// TIA Portal V20 export
// export: Created 2026-09-14T11:29:01.3083632Z, ExportSetting None, DisplayName Totally Integrated Automation Portal, DisplayVersion V20, DisplayName TIA Portal Openness, DisplayVersion V20, DisplayName TIA Portal Version Control Interface, DisplayVersion V20, DisplayName STEP 7 Professional, DisplayVersion V20, DisplayName STEP 7 Safety, DisplayVersion V20, DisplayName WinCC Basic/Comfort/Advanced, DisplayVersion V20, DisplayName WinCC Unified, DisplayVersion V20
TYPE "LMQTT_typeSubscriptionData"
   STRUCT
      newMessageRecieved : Bool;   // Is TRUE for one cycle to signal that new data was recieved
      messageInvalid : Bool;   // Is TRUE, when either internal Buffer of FB is too small or recieved Message Data string length is too low
      receivingTopic : WString[300];   // The topic for which the message was recieved
      receivedMessageData : WString[1450];   // The received data (payload)
   END_STRUCT;
END_TYPE
